(* IEC 61131-3 sources: pen-manipulator/, 13 files *)

(* ---- PathPoint.st ---- *)
//
// Describes a single entry in a motion path.
// P1 and P3 define the start and end points of the move.
// P2 is used for intermediate information: it is the end point when
// `IsArc` is FALSE or the mid point of an arc when `IsArc` is TRUE.
//
TYPE PathPoint :
STRUCT
    P1 : POS2D; // Start point
    P2 : POS2D; // Midpoint for arc or endpoint for line
    P3 : POS2D; // Endpoint for arc (ignored for line)
    IsArc : BOOL;
    Break : BOOL; // If TRUE, stop after this segment
END_STRUCT
END_TYPE

(* ---- Pos2D.st ---- *)
TYPE Pos2D :
STRUCT
	X : REAL;
    Y : REAL;
END_STRUCT
END_TYPE

(* ---- FU_atan2.st ---- *)
//
// Basic implementation of the mathematical ATAN2 function.  It returns
// the angle of the vector (x, y) in radians and mirrors the behaviour of
// the standard C function of the same name.
//
FUNCTION FU_atan2 : REAL
VAR_INPUT
    y : REAL;
    x : REAL;
END_VAR
VAR
    result : REAL;
END_VAR

IF x > 0 THEN
    result := ATAN(y / x);
ELSIF x < 0 AND y >= 0 THEN
    result := ATAN(y / x) + 3.1415926;
ELSIF x < 0 AND y < 0 THEN
    result := ATAN(y / x) - 3.1415926;
ELSIF x = 0 AND y > 0 THEN
    result := 3.1415926 / 2;
ELSIF x = 0 AND y < 0 THEN
    result := -3.1415926 / 2;
ELSE
    result := 0.0;
END_IF;
FU_atan2 := result;
// End of FU_atan2
END_FUNCTION

(* ---- FU_CanvasOffset.st ---- *)
//
// Function used to translate coordinates from a local canvas
// reference frame to the global coordinate system.  The output
// is the input position shifted by the offset of the canvas in
// the global frame.
//
FUNCTION FU_CanvasOffset : Pos2D
VAR_INPUT
    Source : Pos2D;      // Position in source coordinate system
    Offset : Pos2D;      // Offset of the canvas origin in source coordinates
END_VAR

FU_CanvasOffset.X := Source.X + Offset.X;
FU_CanvasOffset.Y := Source.Y + Offset.Y;
// End of FU_CanvasOffset

(* ---- FB_CanvasOffset.st ---- *)
//
// Function block to translate coordinates from a source reference
// frame (e.g. visualisation) to a local canvas coordinate system.
// The output is simply the input position shifted by the provided
// offset.
//
FUNCTION_BLOCK FB_CanvasOffset
VAR_INPUT
    Source : Pos2D;      // Position in source coordinate system
    Offset : Pos2D;      // Offset of the canvas origin in source coordinates
END_VAR
VAR_OUTPUT
    Canvas : Pos2D;      // Transformed position relative to canvas origin
END_VAR

Canvas.X := Source.X - Offset.X;
Canvas.Y := Source.Y - Offset.Y;
// End of FB_CanvasOffset

(* ---- FB_CircularMove.st ---- *)
//
// Function block implementing a circular movement from P1 to P3 while
// passing through P2.  The block calculates the centre of the circle and
// generates a velocity vector to follow the arc at a trapezoidal speed
// profile.
//
FUNCTION_BLOCK FB_CircularMove
VAR_INPUT
    P1 : POS2D;             // Start point
    P2 : POS2D;             // Midpoint on arc (used only to determine arc path, not a stop point)
    P3 : POS2D;             // End point
    MaxSpeed : REAL;        // Maximum path speed [mm/s]
    Accel : REAL;           // Angular acceleration [rad/s^2]
    t : REAL;               // Time since start of movement [s]
    DecelerateAtEnd : BOOL; // Whether to decelerate at the end of movement
END_VAR
VAR_OUTPUT
    SpeedX : REAL;          // Current velocity in X direction
    SpeedY : REAL;          // Current velocity in Y direction
END_VAR
VAR
    CenterX, CenterY : REAL;
    Radius : REAL;
    StartAngle, EndAngle : REAL;
    CW : BOOL;

    ArcLength : REAL;
    Dir : REAL;
    DeltaAngle : REAL;
    t_acc : REAL;
    s_acc : REAL;
    s_const : REAL;
    t_const : REAL;
    t_total : REAL;
    s_t : REAL;
    v : REAL;
    Angle : REAL;
	angleP2 : REAL;
    AngularSpeed : REAL;
    t_dec : REAL;

    (* Variables for circle center calculation using perpendicular bisectors *)
    dx12, dy12, dx23, dy23 : REAL;
    M12X, M12Y, M23X, M23Y : REAL;
    RHS1, RHS2, D : REAL;
END_VAR

// Main calculation block: Move from P1 to P3 through P2 along a circular arc

// Calculate circle center using perpendicular bisector intersection
dx12 := P2.X - P1.X;
dy12 := P2.Y - P1.Y;
dx23 := P3.X - P2.X;
dy23 := P3.Y - P2.Y;

// Mid‑points of the two chords
M12X := (P1.X + P2.X) * 0.5;
M12Y := (P1.Y + P2.Y) * 0.5;
M23X := (P2.X + P3.X) * 0.5;
M23Y := (P2.Y + P3.Y) * 0.5;

// Determinant for the 2×2 system
D := dx12 * dy23 - dy12 * dx23;

// Abort if points are collinear (determinant ≈ 0)
IF ABS(D) < 1e‑6 THEN
    SpeedX := 0.0;
    SpeedY := 0.0;
    RETURN;
END_IF;

// Right‑hand sides of the linear equations
RHS1 := dx12 * M12X + dy12 * M12Y;
RHS2 := dx23 * M23X + dy23 * M23Y;

// Intersection of the two perpendicular bisectors → circle centre
CenterX := (RHS1 * dy23 - dy12 * RHS2) / D;
CenterY := (dx12 * RHS2 - RHS1 * dx23) / D;

Radius := SQRT((P1.X - CenterX)*(P1.X - CenterX) + (P1.Y - CenterY)*(P1.Y - CenterY));
StartAngle := FU_atan2(P1.Y - CenterY, P1.X - CenterX);
EndAngle := FU_atan2(P3.Y - CenterY, P3.X - CenterX);

angleP2 := FU_atan2(P2.Y - CenterY, P2.X - CenterX);

// Determine clockwise or counterclockwise direction based on arc passing through P2
IF ((StartAngle < EndAngle) AND (angleP2 > StartAngle) AND (angleP2 < EndAngle)) OR
   ((StartAngle > EndAngle) AND NOT (angleP2 > EndAngle AND angleP2 < StartAngle)) THEN
    CW := FALSE;
ELSE
    CW := TRUE;
END_IF;

// Set direction multiplier: -1 for clockwise, +1 for counterclockwise
IF CW = TRUE THEN
	Dir := -1.0;
ELSE
	Dir := 1.0;
END_IF

// Adjust DeltaAngle for proper arc direction considering CW/CCW
DeltaAngle := EndAngle - StartAngle;
IF DeltaAngle < 0 AND NOT CW THEN
    DeltaAngle := DeltaAngle + 2 * 3.1415926;
ELSIF DeltaAngle > 0 AND CW THEN
    DeltaAngle := DeltaAngle - 2 * 3.1415926;
END_IF;
DeltaAngle := ABS(DeltaAngle);
ArcLength := Radius * DeltaAngle;
t_acc := MaxSpeed / Accel;
s_acc := 0.5 * Accel * t_acc * t_acc;
s_const := ArcLength - 2 * s_acc;

IF s_const < 0 THEN
    t_acc := SQRT(ArcLength / Accel);
    t_const := 0.0;
    t_total := 2 * t_acc;
ELSE
    t_const := s_const / MaxSpeed;
    t_total := 2 * t_acc + t_const;
END_IF;

// Acceleration phase
IF t < t_acc THEN
    v := Accel * t;
    s_t := 0.5 * Accel * t * t;

// Constant speed phase or skipping deceleration
ELSIF t < t_acc + t_const OR NOT DecelerateAtEnd THEN
    v := MaxSpeed;
    s_t := s_acc + v * (t - t_acc);

// Deceleration phase
ELSIF t < t_total THEN
    t_dec := t - t_acc - t_const;
    v := MaxSpeed - Accel * t_dec;
    s_t := s_acc + s_const + MaxSpeed * t_dec - 0.5 * Accel * t_dec * t_dec;

// Motion complete - stop
ELSE
    v := 0.0;
    s_t := ArcLength;
END_IF;

Angle := StartAngle + Dir * (s_t / Radius);
AngularSpeed := v / Radius;
SpeedX := -SIN(Angle) * AngularSpeed * Radius;
SpeedY := COS(Angle) * AngularSpeed * Radius;
// End of FB_CircularMove

(* ---- FB_CircularMovePI.st ---- *)
//
// Circular move using a PI controller. The block keeps track of the current
// angle along the arc and computes a target point on the circle for every
// cycle. The velocity to this target is generated by two PI controllers.
//
FUNCTION_BLOCK FB_CircularMovePI
VAR_INPUT
    CurPos : POS2D;   // Current TCP position
    P1 : POS2D;       // Start point of the arc
    P2 : POS2D;       // Mid point defining the arc
    P3 : POS2D;       // End point of the arc
    MaxSpeed : REAL;  // Desired tangential speed [mm/s]
    Kp : REAL;        // Proportional gain
    Ki : REAL;        // Integral gain
    Ts : REAL;        // Cycle time [s]
END_VAR
VAR_IN_OUT
    SpeedX : REAL;    // Current speed command X (state on call)
    SpeedY : REAL;    // Current speed command Y (state on call)
END_VAR
VAR
    IntX : REAL;
    IntY : REAL;
    CenterX, CenterY : REAL;
    Radius : REAL;
    StartAngle : REAL;
    EndAngle : REAL;
    Angle : REAL;
    Dir : REAL;           // +1 CCW, -1 CW
    InitDone : BOOL := FALSE;
    ErrX, ErrY : REAL;
    TargetX, TargetY : REAL;
    SpeedMag : REAL;

    // Temporary variables for circle calculation
    dx12, dy12, dx23, dy23 : REAL;
    M12X, M12Y, M23X, M23Y : REAL;
    RHS1, RHS2, D : REAL;
    angleP2 : REAL;

    AngleError : REAL;
    AngleInt : REAL;
    AngleKp : REAL := 10.0;
    AngleKi : REAL := 50.0;
END_VAR

IF NOT InitDone THEN
    dx12 := P2.X - P1.X;
    dy12 := P2.Y - P1.Y;
    dx23 := P3.X - P2.X;
    dy23 := P3.Y - P2.Y;

    M12X := (P1.X + P2.X) * 0.5;
    M12Y := (P1.Y + P2.Y) * 0.5;
    M23X := (P2.X + P3.X) * 0.5;
    M23Y := (P2.Y + P3.Y) * 0.5;

    D := dx12 * dy23 - dy12 * dx23;
    IF ABS(D) < 0.0001 THEN
        CenterX := 0.0;
        CenterY := 0.0;
        Radius := 1.0;
    ELSE
        RHS1 := dx12 * M12X + dy12 * M12Y;
        RHS2 := dx23 * M23X + dy23 * M23Y;
        CenterX := (RHS1 * dy23 - dy12 * RHS2) / D;
        CenterY := (dx12 * RHS2 - RHS1 * dx23) / D;
        Radius := SQRT((P1.X - CenterX)*(P1.X - CenterX) + (P1.Y - CenterY)*(P1.Y - CenterY));
    END_IF;

    StartAngle := FU_atan2(P1.Y - CenterY, P1.X - CenterX);
    EndAngle := FU_atan2(P3.Y - CenterY, P3.X - CenterX);
    angleP2 := FU_atan2(P2.Y - CenterY, P2.X - CenterX);

    IF ((StartAngle < EndAngle) AND (angleP2 > StartAngle) AND (angleP2 < EndAngle)) OR
       ((StartAngle > EndAngle) AND NOT (angleP2 > EndAngle AND angleP2 < StartAngle)) THEN
        Dir := 1.0; // CCW
    ELSE
        Dir := -1.0; // CW
    END_IF;

    Angle := StartAngle;
    InitDone := TRUE;
END_IF;

TargetX := CenterX + Radius * COS(Angle);
TargetY := CenterY + Radius * SIN(Angle);

ErrX := TargetX - CurPos.X;
ErrY := TargetY - CurPos.Y;

IntX := IntX + Ki * ErrX * Ts;
IntY := IntY + Ki * ErrY * Ts;

IF IntX > MaxSpeed THEN
    IntX := MaxSpeed;
ELSIF IntX < -MaxSpeed THEN
    IntX := -MaxSpeed;
END_IF;
IF IntY > MaxSpeed THEN
    IntY := MaxSpeed;
ELSIF IntY < -MaxSpeed THEN
    IntY := -MaxSpeed;
END_IF;

SpeedX := Kp * ErrX + IntX;
SpeedY := Kp * ErrY + IntY;

IF SpeedX > MaxSpeed THEN
    SpeedX := MaxSpeed;
ELSIF SpeedX < -MaxSpeed THEN
    SpeedX := -MaxSpeed;
END_IF;
IF SpeedY > MaxSpeed THEN
    SpeedY := MaxSpeed;
ELSIF SpeedY < -MaxSpeed THEN
    SpeedY := -MaxSpeed;
END_IF;

// Use a PI controller to drive the angle progression toward max tangential speed
AngleError := MaxSpeed - SQRT(SpeedX * SpeedX + SpeedY * SpeedY);
AngleInt := AngleInt + AngleKi * AngleError * Ts;
IF AngleInt > MaxSpeed THEN
    AngleInt := MaxSpeed;
ELSIF AngleInt < 0 THEN
    AngleInt := 0;
END_IF;
SpeedMag := AngleKp * AngleError + AngleInt;
IF SpeedMag > MaxSpeed THEN
    SpeedMag := MaxSpeed;
ELSIF SpeedMag < 0 THEN
    SpeedMag := 0;
END_IF;

IF Radius > 0 THEN
    Angle := Angle + Dir * (SpeedMag / Radius) * Ts;
END_IF;

// End of FB_CircularMovePI

(* ---- FB_LinealMove.st ---- *)
//
// Function block implementing a trapezoidal speed profile for linear
// movements.  The block accelerates from the start position, maintains a
// constant speed and optionally decelerates at the end.
//
FUNCTION_BLOCK FB_LinealMove
VAR_INPUT
    StartPos : POS2D;   // Starting position
    TargetPos : POS2D;  // Target position
    MaxSpeed : REAL;    // Maximum speed during movement
    Accel : REAL;       // Acceleration used for ramp-up and ramp-down
    t : REAL;           // Elapsed time since start of movement
    DecelerateAtEnd : BOOL; // Whether to ramp down at the end
END_VAR
VAR_IN_OUT
    SpeedX : REAL;      // Current speed in the X direction (initial value on first call)
    SpeedY : REAL;      // Current speed in the Y direction (initial value on first call)
END_VAR
VAR
    TotalDist : REAL;   // Total distance between start and target
    DirX : REAL;        // Normalized direction vector X component
    DirY : REAL;        // Normalized direction vector Y component
    t_acc : REAL;       // Time needed to accelerate to MaxSpeed
    s_acc : REAL;       // Distance covered during acceleration phase
    s_const : REAL;     // Distance covered at constant MaxSpeed
    t_const : REAL;     // Time spent at constant MaxSpeed
    t_total : REAL;     // Total duration of the entire move
    v : REAL;           // Current magnitude of the velocity vector
    v0 : REAL;          // Initial velocity magnitude
    t_dec : REAL;       // Time needed to decelerate to 0
END_VAR

// Compute direction and total distance
TotalDist := SQRT(EXPT(TargetPos.X - StartPos.X,2) + EXPT(TargetPos.Y - StartPos.Y,2));
IF TotalDist = 0 THEN
    SpeedX := 0;
    SpeedY := 0;
ELSE
    DirX := (TargetPos.X - StartPos.X) / TotalDist;
    DirY := (TargetPos.Y - StartPos.Y) / TotalDist;

    // Determine initial speed magnitude from provided inputs
    v0 := SQRT(SpeedX * SpeedX + SpeedY * SpeedY);

    t_acc := (MaxSpeed - v0) / Accel;
    IF t_acc < 0 THEN
        t_acc := 0;
    END_IF;
    s_acc := v0 * t_acc + 0.5 * Accel * t_acc * t_acc;
    t_dec := MaxSpeed / Accel;
    s_const := TotalDist - s_acc - (0.5 * MaxSpeed * t_dec);

    IF s_const < 0 THEN
        // Triangular profile starting from v0
        v := SQRT(v0 * v0 + 2 * Accel * TotalDist);
        t_acc := (v - v0) / Accel;
        t_dec := v / Accel;
        t_const := 0;
        t_total := t_acc + t_dec;
    ELSE
        // Trapezoidal profile
        t_const := s_const / MaxSpeed;
        t_total := t_acc + t_const + t_dec;
    END_IF;

    // Determine current speed magnitude
    IF t < t_acc THEN
        v := Accel * t;
    ELSIF t < t_acc + t_const OR NOT DecelerateAtEnd THEN
        v := MaxSpeed;
    ELSIF t < t_total THEN
        v := MaxSpeed - Accel * (t - t_acc - t_const);
    ELSE
        v := 0;
    END_IF;

    // Apply speed along direction
    SpeedX := v * DirX;
    SpeedY := v * DirY;
END_IF;

// End of FB_TrapezoidalMove

(* ---- FB_LinealMovePI.st ---- *)
//
// Linear move implemented using two PI controllers operating on the
// X and Y axes. The block drives the TCP towards the provided target
// position and outputs velocity commands saturated to MaxSpeed.
//
FUNCTION_BLOCK FB_LinealMovePI
VAR_INPUT
    CurPos    : POS2D; // Current TCP position
    TargetPos : POS2D; // Target position
    MaxSpeed  : REAL;  // Maximum speed [mm/s]
    Kp        : REAL;  // Proportional gain
    Ki        : REAL;  // Integral gain
    Ts        : REAL;  // Cycle time [s]
END_VAR
VAR_IN_OUT
    SpeedX : REAL; // Current speed command X (state on call)
    SpeedY : REAL; // Current speed command Y (state on call)
END_VAR
VAR
    IntX : REAL;   // Integrator state for X axis
    IntY : REAL;   // Integrator state for Y axis
    ErrX : REAL;
    ErrY : REAL;
END_VAR

ErrX := TargetPos.X - CurPos.X;
ErrY := TargetPos.Y - CurPos.Y;

IntX := IntX + Ki * ErrX * Ts;
IntY := IntY + Ki * ErrY * Ts;

// Anti-windup limits
IF IntX > MaxSpeed THEN
    IntX := MaxSpeed;
ELSIF IntX < -MaxSpeed THEN
    IntX := -MaxSpeed;
END_IF;
IF IntY > MaxSpeed THEN
    IntY := MaxSpeed;
ELSIF IntY < -MaxSpeed THEN
    IntY := -MaxSpeed;
END_IF;

SpeedX := Kp * ErrX + IntX;
SpeedY := Kp * ErrY + IntY;

// Saturate outputs
IF SpeedX > MaxSpeed THEN
    SpeedX := MaxSpeed;
ELSIF SpeedX < -MaxSpeed THEN
    SpeedX := -MaxSpeed;
END_IF;
IF SpeedY > MaxSpeed THEN
    SpeedY := MaxSpeed;
ELSIF SpeedY < -MaxSpeed THEN
    SpeedY := -MaxSpeed;
END_IF;

// End of FB_LinealMovePI

(* ---- FB_PIController.st ---- *)
//
// Simple PI controller used by the motion blocks. Computes an output
// velocity based on the position error. Output and integral are
// clamped to the provided limit to avoid windup.
//
FUNCTION_BLOCK FB_PIController
VAR_INPUT
    Setpoint : REAL;  // Desired value
    Measurement : REAL; // Current value
    Kp : REAL;        // Proportional gain
    Ki : REAL;        // Integral gain
    Ts : REAL;        // Cycle time [s]
    Limit : REAL;     // Maximum absolute output
END_VAR
VAR_IN_OUT
    Integral : REAL;  // Integrator state
END_VAR
VAR_OUTPUT
    Out : REAL;       // Controller output
END_VAR
VAR
    Error : REAL;
END_VAR

Error := Setpoint - Measurement;
Integral := Integral + Ki * Error * Ts;

// Clamp integral term
IF Integral > Limit THEN
    Integral := Limit;
ELSIF Integral < -Limit THEN
    Integral := -Limit;
END_IF;

Out := Kp * Error + Integral;

// Clamp controller output
IF Out > Limit THEN
    Out := Limit;
ELSIF Out < -Limit THEN
    Out := -Limit;
END_IF;

// End of FB_PIController

(* ---- FB_TCPaxes.st ---- *)
//
// Function block implementing a trapezoidal speed profile for linear
// movements.  The block accelerates from the start position, maintains a
// constant speed and optionally decelerates at the end.
//
FUNCTION_BLOCK FB_TCPaxes
VAR_INPUT
	SpeedX : REAL;      // Current speed in the X direction (initial value on first call)
    SpeedY : REAL;      // Current speed in the Y direction (initial value on first call)
END_VAR
VAR_OUTPUT
    rAngle: REAL;          // direction angle
	rAngleX: REAL;
	rAngleY: REAL;
END_VAR

	rAngle := FU_atan2(SpeedY, SpeedX);

	rAngleX:= 50* COS(rAngle); //how much x increases
	rAngleY:= 50* SIN(rAngle); //how much y increases

(* ---- FB_TrapezoidalMove.st ---- *)
//
// Function block implementing a trapezoidal speed profile for linear
// movements.  The block accelerates from the start position, maintains a
// constant speed and optionally decelerates at the end.
//
TYPE POS2D :
STRUCT
    X : REAL;
    Y : REAL;
END_STRUCT
END_TYPE

FUNCTION_BLOCK
VAR_INPUT
    StartPos : POS2D;   // Starting position
    TargetPos : POS2D;  // Target position
    MaxSpeed : REAL;    // Maximum speed during movement
    Accel : REAL;       // Acceleration used for ramp-up and ramp-down
    t : REAL;           // Elapsed time since start of movement
    DecelerateAtEnd : BOOL;
END_VAR
VAR_OUTPUT
    SpeedX : REAL;      // Current speed in the X direction
    SpeedY : REAL;      // Current speed in the Y direction
END_VAR
VAR
    TotalDist : REAL;   // Total distance between start and target
    DirX : REAL;        // Normalized direction vector X component
    DirY : REAL;        // Normalized direction vector Y component
    t_acc : REAL;       // Time needed to accelerate to MaxSpeed
    s_acc : REAL;       // Distance covered during acceleration phase
    s_const : REAL;     // Distance covered at constant MaxSpeed
    t_const : REAL;     // Time spent at constant MaxSpeed
    t_total : REAL;     // Total duration of the entire move
    v : REAL;           // Current magnitude of the velocity vector
END_VAR

// Compute direction and total distance
TotalDist := SQRT((TargetPos.X - StartPos.X)**2 + (TargetPos.Y - StartPos.Y)**2);
IF TotalDist = 0 THEN
    SpeedX := 0;
    SpeedY := 0;
ELSE
    DirX := (TargetPos.X - StartPos.X) / TotalDist;
    DirY := (TargetPos.Y - StartPos.Y) / TotalDist;

    t_acc := MaxSpeed / Accel;
    s_acc := 0.5 * Accel * t_acc * t_acc;
    s_const := TotalDist - 2 * s_acc;
    IF s_const < 0 THEN
        // Triangular profile
        t_acc := SQRT(TotalDist / Accel);
        t_const := 0;
        t_total := 2 * t_acc;
    ELSE
        // Trapezoidal profile
        t_const := s_const / MaxSpeed;
        t_total := 2 * t_acc + t_const;
    END_IF;

    // Determine current speed magnitude
    IF t < t_acc THEN
        v := Accel * t;
    ELSIF t < t_acc + t_const THEN
        v := MaxSpeed;
    ELSIF t < t_total THEN
        v := MaxSpeed - Accel * (t - t_acc - t_const);
    ELSE
        v := 0;
    END_IF;

    // Apply speed along direction
    SpeedX := v * DirX;
    SpeedY := v * DirY;
END_IF;
END_FUNCTION_BLOCK

// End of FB_TrapezoidalMove

(* ---- PLC_PRG.st ---- *)
PROGRAM PLC_PRG
VAR
    // Local TCP position measured from the first path point
    TCPRel : Pos2D := (X:=0.0, Y:=0.0);
    // Absolute TCP position used for distance checks
    TCPAbs : Pos2D := (X:=0.0, Y:=0.0);
    // Integer coordinates for the visualization
    VisuPosX : INT := 0;                // X position in pixels
    VisuPosY : INT := 0;                // Y position in pixels
    // Diameter of the circle used to draw the TCP
    CircleWidth : REAL := 10.0;
    // Flag used to trigger reset on startup
    InitDone : BOOL := FALSE;

    // Absolute destination of the current segment
    Target : Pos2D := (X:=0.0, Y:=0.0);

    cycle_time : REAL := 0.001; // Simulation step time
    MaxSpeed : REAL := 15.0;
    // Gains for the PI controllers
    Kp : REAL := 2.0;
    Ki : REAL := 0.0;
    // Current velocity components used by the motion function blocks
    CurSpeedX : REAL := 0.0;
    CurSpeedY : REAL := 0.0;

    MotionActive : BOOL := TRUE;
    Reset : BOOL := FALSE;

    Path : ARRAY[1..3] OF PathPoint := [
        (P1:=(X:=139.0, Y:=82.0), P2:=(X:=239.0, Y:=82.0), P3:=(X:=239.0, Y:=82.0), IsArc:=FALSE, Break:=FALSE),
        (P1:=(X:=239.0, Y:=82.0), P2:=(X:=364.0, Y:=182.0), P3:=(X:=239.0, Y:=282.0), IsArc:=TRUE, Break:=TRUE),
		(P1:=(X:=239.0, Y:=282.0), P2:=(X:=139.0, Y:=82.0), P3:=(X:=139.0, Y:=82.0), IsArc:=FALSE, Break:=TRUE)
    ];
    CurrentIndex : INT := 1;
    PathLength : INT := 3;
    MovePI : FB_LinealMovePI;
    ArcPI : FB_CircularMovePI;
    // Absolute position of the canvas origin in the global frame
    CanvPos : Pos2D := (X:=226.0, Y:=132.0);
    // Temporary storage for path points converted to global coordinates
    CanvasP1 : Pos2D;
    CanvasP2 : Pos2D;
    CanvasP3 : Pos2D;
    // Flag used when returning to the origin
    Go2Canvas : BOOL := FALSE;
    ReturnHome : BOOL := FALSE;
    ReturnStart : Pos2D;
    HomePos : Pos2D := (X:=25.0, Y:=150.0);
END_VAR

// Automatic reset on first cycle
IF NOT InitDone THEN
    Reset := TRUE;
    InitDone := TRUE;
END_IF;

// Reset position and initialise offsets
IF Reset THEN
    // TCP starts at the home position in absolute coordinates
    TCPAbs := HomePos;
    // No displacement in the local frame at reset
    TCPRel.X := 0.0;
    TCPRel.Y := 0.0;

    // Initialise the visualisation values
    VisuPosX := TO_INT(TCPRel.X - CircleWidth / 2.0);
    VisuPosY := TO_INT(TCPRel.Y - CircleWidth / 2.0);
    // Reset velocity
    CurSpeedX := 0.0;
    CurSpeedY := 0.0;
    CurrentIndex := 1;
    ReturnHome := FALSE;
    Go2Canvas := TRUE;
    Reset := FALSE;
END_IF

// Control movement execution
IF MotionActive THEN
    // First move from outside the Canvas to first canvas point
    IF  NOT ReturnHome and Go2Canvas THEN
        // Convert first path point from canvas to global coordinates
        CanvasP2 := FU_CanvasOffset(Path[1].P1, CanvPos);
        Target := CanvasP2;
        // Move to initial position in canvas
        MovePI(
                CurPos := TCPAbs,
                TargetPos := CanvasP2,
                MaxSpeed := MaxSpeed,
                Ts := cycle_time,
                Kp := Kp,
                Ki := Ki,
                SpeedX := CurSpeedX,
                SpeedY := CurSpeedY
            );

    // Moving throught the canvas path
    ELSIF NOT ReturnHome AND CurrentIndex <= PathLength THEN
        // Convert current path segment to global coordinates
        CanvasP1 := FU_CanvasOffset(Path[CurrentIndex].P1, CanvPos);
        CanvasP2 := FU_CanvasOffset(Path[CurrentIndex].P2, CanvPos);
        CanvasP3 := FU_CanvasOffset(Path[CurrentIndex].P3, CanvPos);

        IF NOT Path[CurrentIndex].IsArc THEN
            // Handle linear motion segments using PI control
            MovePI(
                CurPos := TCPAbs,
                TargetPos := CanvasP2,
                MaxSpeed := MaxSpeed,
                Kp := Kp,
                Ki := Ki,
                Ts := cycle_time,
                SpeedX := CurSpeedX,
                SpeedY := CurSpeedY
            );
            Target := CanvasP2;
        ELSE
            // Handle arc-based motion segments using PI control
            ArcPI(
                CurPos := TCPAbs,
                P1 := CanvasP1,
                P2 := CanvasP2,
                P3 := CanvasP3,
                MaxSpeed := MaxSpeed,
                Kp := Kp,
                Ki := Ki,
                Ts := cycle_time,
                SpeedX := CurSpeedX,
                SpeedY := CurSpeedY
            );
            Target := CanvasP3;
        END_IF
    ELSIF ReturnHome THEN
        // Move back to the home position after completing the path
        MovePI(
            CurPos := TCPAbs,
            TargetPos := HomePos,
            MaxSpeed := MaxSpeed,
            Kp := Kp,
            Ki := Ki,
            Ts := cycle_time,
            SpeedX := CurSpeedX,
            SpeedY := CurSpeedY
        );
        Target := HomePos;
    END_IF
    // Integrate velocity to update position
    TCPAbs.X := TCPAbs.X + CurSpeedX * cycle_time;
    TCPAbs.Y := TCPAbs.Y + CurSpeedY * cycle_time;
    // Update relative coordinates after integrating
    TCPRel.X := TCPAbs.X - HomePos.X;
    TCPRel.Y := TCPAbs.Y - HomePos.Y;

    // Convert precise position to integer for visualization
    VisuPosX := TO_INT(TCPRel.X - CircleWidth / 2.0);
    VisuPosY := TO_INT(TCPRel.Y - CircleWidth / 2.0);

    // Check if current target is reached and progress to next segment
    IF ABS(TCPAbs.X - Target.X) < 1 AND ABS(TCPAbs.Y - Target.Y) < 1 THEN
        IF Go2Canvas THEN
            Go2Canvas := FALSE;
        ELSE
            CurrentIndex := CurrentIndex + 1;
        END_IF

        IF CurrentIndex > PathLength AND NOT ReturnHome THEN
            // Begin return to origin on completion
            ReturnHome := TRUE;
            ReturnStart := TCPRel;
        END_IF;
        IF ReturnHome THEN
            // Set target to home position for return
            Target := HomePos;
            MotionActive := FALSE;
            ReturnHome := FALSE;
        END_IF;
    END_IF;
END_IF;

// End of PLC_PRG
